TYPE ST_ColorCMYK :
STRUCT
	nCyan						: BYTE;
	nMagenta					: BYTE;
	nYellow						: BYTE;
	nKey						: BYTE;
END_STRUCT
END_TYPE

(* stored: Version 1.1.0.1
   DUT ST_ColorCMYK: Id {f5aa018c-e9d5-4c30-88f3-f5983a42ee5b} *)
